FUNCTION InRange : BOOL
VAR_INPUT
	v1 : LREAL;
	v2 : LREAL;
	value : LREAL;
	
	inclusive : BOOL;
END_VAR
VAR
	lower : LREAL;
	upper : LREAL;
END_VAR

lower := MIN(v1, v2);
upper := MAX(v1, v2);

IF inclusive THEN
	InRange := (value >= lower AND value <= upper);
ELSE
	InRange := (value > lower AND value < upper);
END_IF

END_FUNCTION

(* stored: Version 1.1.0.1, ProductVersion 3.1.4024.11
   POU InRange: Id {67a1dc66-fa74-417f-82b2-d5cf0e606fd4}, SpecialFunc None *)
